INTERFACE I_QuantityINTPublic EXTENDS I_QuantityPublic, I_QuantityINT


PROPERTY Val : INT
SET
END_SET
END_PROPERTY

END_INTERFACE

(* stored: Version 1.1.0.1
   Itf I_QuantityINTPublic: Id {e7fa7469-c069-418d-bb6f-524f2b84f173}
   Property Val: Id {694b2bda-9c0a-4684-acf8-e024e150e79c}
   Set Set: Id {1c971d17-99ee-4619-a1ea-f47cfb171139} *)
